FUNCTION_BLOCK Fb2PosControl //Регулятор двухпозиционный.

//       Db2PosControl
//     +---------------+
//     | Fb2PosControl |
//  ->-|PV           OP|->-
//    -|SP             |
//    -|HYST           |
//     +---------------+

VAR_INPUT //Входные переменные, сохраняемые.
PV   :REAL := 0.0; //Измеренное значение регулируемого параметра.
SP   :REAL := 0.0; //Заданное значение регулируемого параметра.
HYST :REAL := 5.0; //Гистерезис > 0.
END_VAR

VAR_OUTPUT //Выходные переменные, сохраняемые.
OP :BOOL := FALSE; //Выход управляющего сигнала.
END_VAR

VAR //Внутренние переменные, сохраняемые.
ER :REAL := 0.0; //Ошибка регулирования.
END_VAR

//Ошибка регулирования.
ER := SP - PV;

//Регулятор двухпозиционный.
IF (ER >= HYST)
THEN
OP:=TRUE;
END_IF;

IF (ER <= HYST * (-1.0))
THEN
OP := FALSE;
END_IF;

END_FUNCTION_BLOCK

//Применение.
//
//Двухпозиционный регулятор используется как простейший регулятор температуры, давления, уровня.

// Условное графическое обозначение.
//
//      +---------------+
//      |               |
//      |    +--<--+--  |
//      |    |     |    |
// ER->-|    v     ^    |->-OP
//      |    |     |    |
//      |  --+-->--+    |
//      |               |
//      +---------------+

// Статическая характеристика.
//
//                 OP
//                  ^
//                  |
//           ***<***1***<******
//           *      |      *
//           v      |      ^
//           *      |      *
// -ER <--******>***0***>***--> +ER
//           |      |      |
//           |<---->|<---->|
//             HYST   HYST

// Временная характеристика.
//
// ^ PV,SP
// |         PV
// |----------*---------------*------
// |         * *             * *   |
// |        *   *           *   *  |  SP + HYST
// |       *     *         *       |
// |======*=======*=======*========== SP
// |     *         *     *         |
// |    *           *   *          |  SP - HYST
// |   *             * *           |
// |--*---------------*--------------
// | *
// |*
// +-----------------------------------------> t[s]
//
// ^ OP
// |
// 1***********       *********
// |          *       *       *
// 0----------*********-------***------------> t[s]

// Схема включения.
//
//                  +---------------+
//                  |               |   Объект управления
//                  |    +--<--+--  |     +-----------+
//        +---+ ER  |    |     |    | OP  |     K     |
// SP-->--| + |-->--|    v     ^    |-->--| --------- |-->--+-->PV
// PV  +--| - |     |    |     |    |     | T * s + 1 |     |
//     |  +---+     |  --+-->--+    |     +-----------+     |
//     |            |               |                       |
//     |            +---------------+                       |
//     |                                                    |
//     +----------------------------------------------------+

//  +---------+
//  | GNU GPL |
//  +---------+
//  |
//  |
//  .= .-_-. =.
// ((_/)o o(\_))
//  `-'(. .)`-'
//  |/| \_/ |\
//  ( |     | )
//  /"\_____/"\
//  \__)   (__/
